PROGRAM Shutdown
VAR
	bStart	AT%I* : BOOL := FALSE;
	Shutdown_Block: NT_Shutdown;
END_VAR

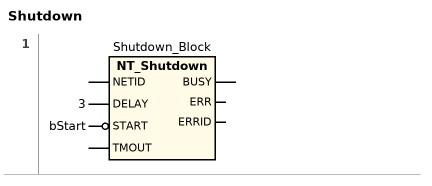
// NETWORK 1
Shutdown_Block(DELAY := 3, START := NOT bStart); // NT_Shutdown

END_PROGRAM

(* stored: Version 1.1.0.1, ProductVersion 3.1.4022.3
   POU Shutdown: Id {037c1cb7-3ef3-4dd0-85e7-d9b82fc4838a}, SpecialFunc None *)
